SUBAPPLICATION Uebung_215_AI (* Standard IEC 61131-3 AI_FB_CTD (Adapter Version, Rückwärtszähler, INT) mit Terminal-Ausgabe *)
  (* Standard: 61131-3; Description: Copyright (c) 2026 Meisterschulen am Ostbahnhof This program and the accompanying materials are made available under the terms of the Eclipse Public License 2.0 which is available at https://www.eclipse.org/legal/epl-2.0/ SPDX-License-Identifier: EPL-2.0 *)
  (* Version 1.2, 2026-05-13, Franz Höpfinger, Meisterschulen am Ostbahnhof, Added AI_INT_TO_I init block connected to PV *)
  (* Version 1.1, 2026-04-21, Franz Höpfinger, Meisterschulen am Ostbahnhof, Added terminal output for counter value *)
  (* Version 1.0, 2026-04-21, Franz Höpfinger, Meisterschulen am Ostbahnhof, initial API and implementation (Adapter version) *)
  PACKAGE Uebungen;
  IMPORT Uebungen::const::UT::DefaultPool::OutputNumber_N1;
  IMPORT logiBUS::io::DI::logiBUS_DI::Input_I1;
  IMPORT logiBUS::io::DI::logiBUS_DI::Input_I2;
  IMPORT logiBUS::io::DQ::logiBUS_DO::Output_Q1;
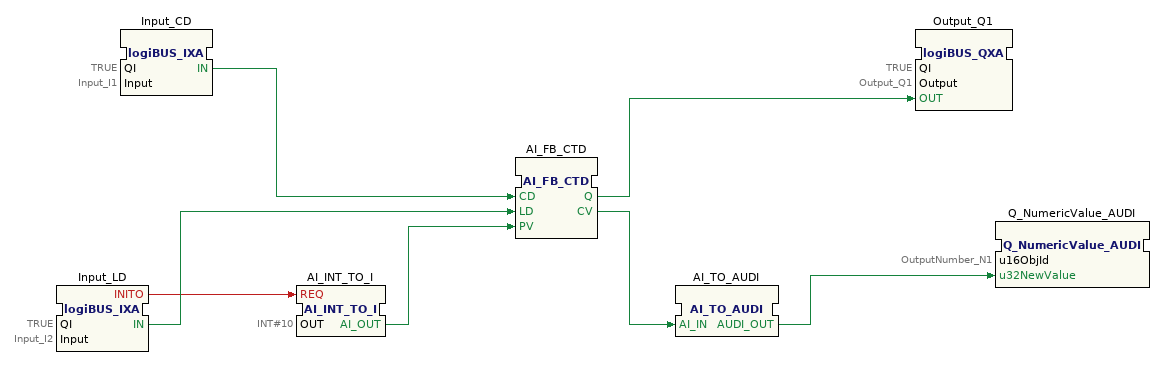
  (* AI_TO_AUDI ist großer Quatsch ... keine Negativen Zahlen möglich *)
  (* hier gegebenenfalls einen AX_D_FF einbauen, damit die Events reduziert werden. *)
  FBS
    AI_FB_CTD : adapter::iec61131::counters::AI_FB_CTD;
    AI_INT_TO_I : adapter::conversion::unidirectional::AI_INT_TO_I(OUT := INT#10);
    Input_CD : logiBUS::io::DI::logiBUS_IXA(QI := TRUE, Input := Input_I1);
    Input_LD : logiBUS::io::DI::logiBUS_IXA(QI := TRUE, Input := Input_I2);
    Output_Q1 : logiBUS::io::DQ::logiBUS_QXA(QI := TRUE, Output := Output_Q1);
    AI_TO_AUDI : adapter::conversion::unidirectional::AI_TO_AUDI;
    Q_NumericValue_AUDI : isobus::UT::Q::Q_NumericValue_AUDI(u16ObjId := OutputNumber_N1);
  END_FBS
  EVENT_CONNECTIONS
    Input_LD.INITO TO AI_INT_TO_I.REQ;
  END_CONNECTIONS
  ADAPTER_CONNECTIONS
    Input_CD.IN TO AI_FB_CTD.CD;
    Input_LD.IN TO AI_FB_CTD.LD;
    AI_FB_CTD.Q TO Output_Q1.OUT;
    AI_FB_CTD.CV TO AI_TO_AUDI.AI_IN;
    AI_TO_AUDI.AUDI_OUT TO Q_NumericValue_AUDI.u32NewValue;
    AI_INT_TO_I.AI_OUT TO AI_FB_CTD.PV;
  END_CONNECTIONS
END_SUBAPPLICATION
